Universal Robots URScript: test2.urscript

def test():

movej([0, -0.94247779, 0, -0.94247779, 0, 0],a=0.1,v=0.05)

end
